Yaskawa INFORM job: M010OPEN.JBI

/JOB
//NAME M010OPEN
//POS
///NPOS 0,0,0,0,0,0
//INST
///DATE 2019/08/05 22:05
///ATTR SC,RW
///GROUP1 RB1
///LVARS 0,0,3,0,0,0,0,0
NOP
SET B069 0
SKILLSND "Comm011Open"
WAIT B069=1
END
